FUNCTION_BLOCK FB_HE_SATT_FilterHolderSelector IMPLEMENTS I_HE_SATT_FilterHolderSelector
VAR
    abSelectedHolder : ARRAY[1..PL_HE_SATT_Parameters.nNumHolders] OF BOOL;
    abCoupledHolders : ARRAY[1..PL_HE_SATT_Parameters.nNumHolders] OF BOOL;
END_VAR


METHOD CoupleHolders
VAR_INPUT
	abCoupledHolders : ARRAY [1..PL_HE_SATT_Parameters.nNumHolders] OF BOOL;
END_VAR

THIS^.abCoupledHolders := abCoupledHolders;
END_METHOD


METHOD CouplingRulesSatisfied : BOOL
VAR_INPUT
	iFilterCombination	: I_HE_SATT_FilterCombination;
END_VAR
VAR
    abFilterHolderIsUsed : ARRAY[1..PL_HE_SATT_Parameters.nNumHolders] OF BOOL;
    nIteratorHolder : INT;
    iFilter : I_HE_SATT_Filter;
    bStateAllCoupledHoldersNeedToBeIn : BOOL;
END_VAR

CouplingRulesSatisfied := TRUE;

FOR nIteratorHolder := 1 TO PL_HE_SATT_Parameters.nNumHolders BY 1 DO
    iFilter := iFilterCombination.GetFilter(nIteratorHolder);
    
    abFilterHolderIsUsed[nIteratorHolder] := iFilter <> 0;
    
    IF THIS^.abCoupledHolders[nIteratorHolder] THEN
        bStateAllCoupledHoldersNeedToBeIn := abFilterHolderIsUsed[nIteratorHolder];
    END_IF
END_FOR

FOR nIteratorHolder := 1 TO PL_HE_SATT_Parameters.nNumHolders BY 1 DO
    IF THIS^.abCoupledHolders[nIteratorHolder] THEN
        CouplingRulesSatisfied := CouplingRulesSatisfied AND (NOT bStateAllCoupledHoldersNeedToBeIn XOR abFilterHolderIsUsed[nIteratorHolder]);
    END_IF
END_FOR
END_METHOD


METHOD DeselectHolder
VAR_INPUT
	nHolderNumber	: INT;
END_VAR

THIS^.abSelectedHolder[nHolderNumber] := FALSE;
END_METHOD


METHOD IsSelected : BOOL
VAR_INPUT
	nHolderNumber	: INT;
END_VAR

IsSelected := THIS^.abSelectedHolder[nHolderNumber];
END_METHOD


METHOD Reset
VAR
    nIteratorHolder : INT;
END_VAR

FOR nIteratorHolder := 1 TO PL_HE_SATT_Parameters.nNumHolders BY 1 DO
    THIS^.abSelectedHolder[nIteratorHolder] := FALSE;
END_FOR
END_METHOD

{warning 'Add method implementation '}
METHOD SelectAll
END_METHOD


METHOD SelectHolder
VAR_INPUT
	nHolderNumber	: INT;
END_VAR

THIS^.abSelectedHolder[nHolderNumber] := TRUE;
END_METHOD

END_FUNCTION_BLOCK

(* stored: Version 1.1.0.1
   POU FB_HE_SATT_FilterHolderSelector: Id {2aa7d618-8dc5-44ab-8dfd-b1f90d9e21ac}, SpecialFunc None
   Method CoupleHolders: Id {2ba254ab-3943-4c44-aafc-e60244281d4f}
   Method CouplingRulesSatisfied: Id {b387d435-f96f-4411-a3bf-4daf2d4804b8}
   Method DeselectHolder: Id {9c8ce84f-c16b-4dca-9baf-bb8ac0752ff9}
   Method IsSelected: Id {4894af9d-86ba-4fdf-9e41-70bce879ed0f}
   Method Reset: Id {f9233bc3-1986-4c92-9e64-727d67abab59}
   Method SelectAll: Id {efc2ff49-45da-47c6-99ae-999f156848e2}
   Method SelectHolder: Id {1b971a68-1703-40cb-8b9c-8965d67e9a05} *)
